(* CODESYS project CtaAppDumper_2.0.0.0.library
   Description: Dumper Library der CTA
   Version: 2.0.0.0
   Title: CtaAppDumper
   Author: SIS
   DocFormat: reStructuredText
   LanguageModelAttribute: qualified-access-only
   Placeholder: CtaAppDumper
   CompiledLibraryCompatibilityVersion: CODESYS V3.5 SP16 Patch 3
   Company: CTA
   DefaultNamespace: CtaAppDumper

Project tree, tasks and I/O mapping:
  libraries: CtaSysConfig, 2.0.0.0 (CTA); CtaAppTime, 1.0.0.1 (CTA); CtaVisSymbols, 2.0.0.0 (CTA); VisuSymbols, 4.5.0.0 (System)
  40 Visualizations/
    visualisation visDumper
    visualisation visPopUpDumper
    visualisation VisDumperSmall
  30 Program Organization Units/
    function block fbDumper [ST]: actConfigFile
  00000000-0000-0000-0000-000000000000|D:\CoDeSys\LibrariesV3\trunk\Intern\CAA\CAA Template\3.4.0.0 draft\Placeholder.xml
  00000000-0000-0000-0000-000000000000|D:\CoDeSys\LibrariesV3\trunk\Intern\CAA\CAA Template\3.2.0.3 draft\Prefix.pdf
  00000000-0000-0000-0000-000000000000|D:\CoDeSys\LibrariesV3\trunk\Intern\CAA\CAA Template\3.5.2.0 draft\Placeholder.xml
  20 Structs/
    data type scParameter
  50 Images/
  10 Documenation/
    global variables VersionHistory
    global variables readMe
  21 Interface/
  11 Library Parameter/
  12 Konstanten/
  60 Textlisten/
  13 Globale Variablen/
  text list GlobalTextList
*)

// 20 Structs/scParameter
TYPE scParameter :
	STRUCT
		fbrTup      		:	CtaSysConfig.fbREAL;	// Erhöung um Referenzwert                                         
    	fbrTdown    		:	CtaSysConfig.fbREAL;	// Verminderung um Referenzwert                                    
   		fbrBand     		:	CtaSysConfig.fbREAL;	// Referenz wert welcher in der Zeit Tup oder Tdown integriert wird
   		fbxInExpOut 		:	CtaSysConfig.fbBOOL;	// rSoll = rY wenn xEn False                                       
	END_STRUCT
END_TYPE

// 10 Documenation/VersionHistory
(* 

.. image:: ../../Images/CTA_Logo.jpg
   :align: right
   :width: 15% 

**Vorlage**   


============ =========== =========== ============================================
**Date**     **Version** **Author**  **Change**
------------ ----------- ----------- --------------------------------------------
04.03.2021   0.0.0.0     SIS         Vorlage erstellt

============ =========== =========== ============================================


*)
VAR_GLOBAL
    stInfo : STRING:= '0.0.0.0, Vorlage, CTA';
END_VAR

// 10 Documenation/readMe
(*

**ReadMe**
 
|	**Empfehlung**
|
|	Bibliothek CtaAppDumper zur dämpfung und rampung von Signalen
|	Instanzieren Sie den CtaAppDumper.fbDumper in ihrem Funktionsbaustein oder POU beispielsweise als fbVerdichterRampe 
|	Deklarieren Sie die Struktur Variable welche als Parameter und zur ansteuerung dienen wie im Code beispiel.
|  
| *Beispiel* 

+-----------------------+---------------------------------------------------------------------------------------------------------------------------------------------------------------------------------------------------------------------------------------------------------------------------------------------------------------------------------------------------------------------------------------------------------------------------------------+
| Beschreibung          |  Code                                                                                                                                                                                                                                                                                                                                                                                                                                 |
+=======================+=======================================================================================================================================================================================================================================================================================================================================================================================================================================+
| POU oder SmFb         | .. code-block:: codesys                                                                                                                                                                                                                                                                                                                                                                                                               |
|                       |                                                                                                                                                                                                                                                                                                                                                                                                                                       |
|                       |	// Deklaration als VAR im POU oder dem selbsterstellten Funktionsbaustein                                                                                                                                                                                                                                                                                                                                                        	|
|                       |   VAR   																																																				 																																																				|
|						|	    (*Verdichter Rampe 1*)																																																		 																																																	|
|						|		fbVerdichterRampe			: CtaAppDumper.fbDumper;																																																																																											|
|			 			|	END_VAR                                                                                                                                                                                                                                                                                                                                                                                                                          	|
+-----------------------+---------------------------------------------------------------------------------------------------------------------------------------------------------------------------------------------------------------------------------------------------------------------------------------------------------------------------------------------------------------------------------------------------------------------------------------+
| Code für Init         | .. code-block:: codesys                                                                                                                                                                                                                                                                                                                                                                                                               |
|                       |   																																																					 																																																				|
|			 			|	// Kopieren des nachfolgenden Codes in eine Action zur Initialisierung der Parameter. Zum Beispiel actConfig.																																																				 																										|
|                       |	{region "Parameter Temperaturfühler 1"}                                                                                                                                                                                                                                                                                                                                                                                             |
|			 			|		(*Basis*)                                                                                                                                                                                                                                                                                                                                                                                                                       |
|						|		fbVerdichterRampe.scParameter.fbrTup					(_WertInit :=	300				, _MinInit :=			, _MaxInit :=			);     //P2 Vorgabe für das Hochrampen																																																													|
|						|		fbVerdichterRampe.scParameter.fbrTdown					(_WertInit :=	 80				, _MinInit :=			, _MaxInit :=			);     //P3 Vorgabe für das Runterrampen																																																												|
|						|		fbVerdichterRampe.scParameter.fbrBand					(_WertInit :=   100				, _MinInit :=			, _MaxInit :=			);     //P4 Band für die Rampung																																																														|
|						|		fbVerdichterRampe.scParameter.fbxInExpOut				(_WertInit := FALSE																);     //P5 In = Out wenn True																																																															|
|						|	{endregion}                                                                                                                                                      																																																																    | 
|						|																																																																																																										|
+-----------------------+---------------------------------------------------------------------------------------------------------------------------------------------------------------------------------------------------------------------------------------------------------------------------------------------------------------------------------------------------------------------------------------------------------------------------------------+
*)                                                                                                                                                                                                                                                                                                                                                                                                                                                               
VAR_GLOBAL
	xReadMeDone              :   BOOL; 
END_VAR

// 30 Program Organization Units/fbDumper
//*******************************************************************************************************************************************************************************************************************************************//
//  Author:         SIS                                                                           																																			 //
//  Version:        1.0.0.0		                                                                      																																		 //
//  Beschreibung:   Dumper                                                                       																																			 //
//                                                                          																										                                                	     //
//                                                                             																						 				                                                		 //
//                                                                             																										                                                	  	 //
//*******************************************************************************************************************************************************************************************************************************************//
FUNCTION_BLOCK fbDumper
//===========================================================================================================================================================================================================================================//
//  Variabeln Deklaration  Input                                                                  																																			 //
//===========================================================================================================================================================================================================================================//
VAR_INPUT   
    xEn             :   BOOL;                                                                    // Regler Freigabe                                            
    rSoll           :   REAL;                                                                    // Sollwert    
END_VAR
//===========================================================================================================================================================================================================================================//
//  Variabeln Deklaration  Output                                                                																																			 //
//===========================================================================================================================================================================================================================================//
VAR_OUTPUT                      
    rY				:	REAL;                                   // Die Stellgrösse Y am Ausgang
END_VAR

VAR
    scParameter		:	scParameter;
    rIntegral		:	REAL;                                   // Integrationswert
    rCycleTime		:	REAL;                                   // Zylkuszeit
    xRelease		:	BOOL;    
    fbCycle			:  	CtaAppTime.fbTimeMeasurement ;
	fbConfigFile    :   CtaSysConfig.fbConfigFile;		       // ConfigFile Fb
END_VAR

//===========================================================================================================================================================================================================================================//
//  Config File                                                                                  																																			 //
//===========================================================================================================================================================================================================================================//
actConfigFile();
//===========================================================================================================================================================================================================================================//
//  Freigabe des Regler über die Funktion xEN                                                                                                                                                                                                //
//===========================================================================================================================================================================================================================================//
// Zykluszeit erkennen
rCycleTime  :=  LTIME_TO_REAL(fbCycle.stop())/1000000000; // Ltime to ms
fbCycle.Start();
IF xEn THEN
    (* Wertüberwachung *)
    IF scParameter.fbrTup.proValue <= 0 THEN
        scParameter.fbrTup.proValue := 0.1;
	END_IF
    (* Wertüberwachung *)
    IF scParameter.fbrTdown.proValue <= 0 THEN
        scParameter.fbrTdown.proValue := 0.1;
	END_IF;
    IF (rSoll > rY) THEN
        IF (scParameter.fbrTup.proValue > 0) THEN 
            IF rCycleTime > 0 THEN
                rIntegral := ((scParameter.fbrBand.proValue/ scParameter.fbrTup.proValue) * rCycleTime); 
            END_IF;
            IF (rSoll - rY) < rIntegral THEN
                // Ausgangswert Zusammengesetzt aus Stellwert und Integrationswert
                rY := (rY +  (rSoll-rY));
                
            ELSE              
                // Ausgangswert Zusammengesetzt aus Stellwert und Integrationswert
                rY := (rY + rIntegral);
                
            END_IF;
        END_IF;
    ELSIF  (rSoll < rY) THEN  
        IF scParameter.fbrTdown.proValue > 0 THEN 
            IF rCycleTime > 0 THEN
            rIntegral := ((scParameter.fbrBand.proValue/ scParameter.fbrTdown.proValue) * rCycleTime); 
            END_IF;
            IF (rY-rSoll) < rIntegral THEN
                // Ausgangswert Zusammengesetzt aus Stellwert und Integrationswert
                rY := (rY -  (rY-rSoll));
            ELSE
                // Ausgangswert Zusammengesetzt aus Stellwert und Integrationswert
                rY := (rY -  rIntegral);
            END_IF;
        END_IF;
    ELSIF rSoll = rY THEN
        rY:= rY;
    END_IF;   
//===========================================================================================================================================================================================================================================//
//  Wertverhalten bei Not xEN                                                                                                                                                                                                                //
//===========================================================================================================================================================================================================================================//         
ELSIF (NOT xEn) THEN
    IF scParameter.fbxInExpOut.proValue THEN
        rY  :=  rSoll;
    ELSE    
        rY  :=  0.0;
    END_IF;     
END_IF;

ACTION actConfigFile:
// Aufruf fbConfigFile
fbConfigFile();
(* Aufruf der Parameter Bausteine in Fb*)
scParameter.fbrTup		(_usiParaNr := 1 , itfConfigFb := fbConfigFile);
scParameter.fbrTdown	(_usiParaNr := 2 , itfConfigFb := fbConfigFile);
scParameter.fbrBand		(_usiParaNr := 3 , itfConfigFb := fbConfigFile);
scParameter.fbxInExpOut	(_usiParaNr := 4 , itfConfigFb := fbConfigFile);
END_ACTION

END_FUNCTION_BLOCK

// 40 Visualizations/visDumper
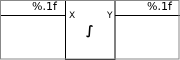
VISUALIZATION visDumper  // 180x60
VAR_IN_OUT
    fbDumper  :   fbDumper;		
END_VAR
    Textfield (0,0 60x13), "%.1f", text variable: fbDumper.rSoll
    Line (0,15) (180,15)
    Textfield (65,0 50x60), "∫"
        OnMouseClick:  Dialog=visPopUpDumper, Parameters={fbDumper: fbDumper}, Selected={0: }, OpenCentered=True
    Label (66,10 20x10), "X"
    Label (104,10 10x10), "Y"
    Textfield (115,0 60x13), "%.1f", text variable: fbDumper.rY
END_VISUALIZATION

// 40 Visualizations/visPopUpDumper
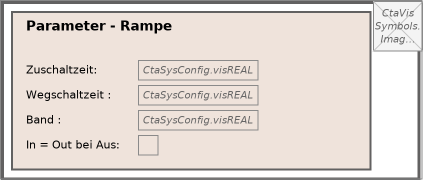
VISUALIZATION visPopUpDumper  // 423x180
VAR_IN_OUT
    fbDumper  :   fbDumper;		
END_VAR
    RoundedRectangle (1,1 419x179)
    RoundedRectangle (11,11 360x159)
    Label (23,60 120x20), "Zuschaltzeit:"
    Label (23,85 120x20), "Wegschaltzeit :"
    Image (373,1 50x50), image: CtaVisSymbols.ImagePool.close_solo_black
        OnMouseClick:  Dialog=visPopUpDumper, Result=None, NumpadKeypadSet=True
    Label (23,110 120x20), "Band :"
    Frame (138,60 120x20)
        shows CtaSysConfig.visREAL(visfbREALIn := fbDumper.scParameter.fbrTup, stPhysikalischeEinheit := 's')
    Frame (138,85 120x20)
        shows CtaSysConfig.visREAL(visfbREALIn := fbDumper.scParameter.fbrTdown, stPhysikalischeEinheit := 's')
    Frame (138,110 120x20)
        shows CtaSysConfig.visREAL(visfbREALIn := fbDumper.scParameter.fbrBand)
    Label (23,135 120x20), "In = Out bei Aus:"
    Frame (138,135 20x20)
        shows CtaSysConfig.visBOOL(visfbBOOLIn := fbDumper.scParameter.fbxInExpOut)
    Label (23,16 150x20), "Parameter - Rampe"
    InvisibleInput (11,1 360x50)
END_VISUALIZATION

// 40 Visualizations/VisDumperSmall
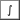
VISUALIZATION VisDumperSmall  // 20x20
VAR_IN_OUT
    fbDumper  :   fbDumper;		
END_VAR
    Textfield (0,0 20x20), "∫"
        OnMouseClick:  Dialog=visPopUpDumper, Parameters={fbDumper: fbDumper}, Selected={0: }, OpenCentered=True
END_VISUALIZATION
